{attribute 'qualified_only'}
{attribute 'strict'}
TYPE JobType :
(
	valid := 0,
	invalid,
	noJob
);
END_TYPE

(* stored: Version 1.1.0.1, ProductVersion 3.1.4024.11
   DUT JobType: Id {497a7a3e-5cda-42b5-b2d6-1c3e4c0929a8} *)
